(* PLC project Projeto_Silos.project, CODESYS CODESYS V3.5 SP11 Patch 4 *)
(* stored: creationDateTime 2025-10-06T19:54:17.7086948, modificationDateTime 2025-10-06T19:50:28.7209293 *)

PROGRAM PLC_PRG

                    
                  
END_PROGRAM

PROGRAM PRG_Simulacao

                    
                  
END_PROGRAM

PROGRAM PRG_Controle

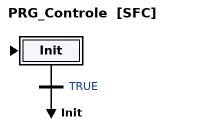
INITIAL_STEP Init:
END_STEP
TRANSITION FROM Init TO Init
  := TRUE;
END_TRANSITION
END_PROGRAM

CONFIGURATION Device
  RESOURCE Application ON PLC
    {attribute 'qualified_only'}
    VAR_GLOBAL  (* GVL_IO *)
      LS_01 : BOOL;  (* Chave fim-de-curso Silo 1. TRUE quando Tripper posicionado. *)
      LS_02 : BOOL;  (* Chave fim-de-curso Silo 2. *)
      LS_03 : BOOL;  (* Chave fim-de-curso Silo 3. *)
      LS_04 : BOOL;  (* Chave fim-de-curso Silo 4. *)
      TR_DIST : REAL;  (* Sensor de distância a laser (metragem) . *)
      WT_01 : REAL;  (* Balança de fluxo interna ao tripper (kg/s) . *)
      TR_FW : BOOL;  (* Acionamento frente do Tripper. *)
      TR_BW : BOOL;  (* Acionamento ré do Tripper. *)
      TR_VEL : REAL;  (* Velocidade de deslocamento do Tripper (m/s) . *)
      M_CT_01 : BOOL;  (* Liga/desliga a correia alimentadora CT-01. *)
      BUZINA : BOOL;  (* Ativa a Buzina para sinalização. *)
    END_VAR
    {attribute 'qualified_only'}
    VAR_GLOBAL  (* GVL_SCADA *)
      LIGA_AUTO : BOOL;  (* Comando de LIGA / DESLIGA executado via SCADA. *)
      EMG : BOOL;  (* Sinalização manual de Emergência via SCADA. *)
      REARME : BOOL;  (* Sinalização manual de Rearme via SCADA. *)
      FV_01 : BOOL;  (* Válvula on-off de descarga Silo 1. *)
      FV_02 : BOOL;  (* Válvula on-off de descarga Silo 2. *)
      FV_03 : BOOL;  (* Válvula on-off de descarga Silo 3. *)
      FV_04 : BOOL;  (* Válvula on-off de descarga Silo 4. *)
      LT_01 : REAL;  (* Sensor de nível Silo 1 (Simulado manualmente via IHM, conforme orientação [cite: 123]). *)
      LT_02 : REAL;  (* Sensor de nível Silo 2 (Simulado manualmente via IHM). *)
      LT_03 : REAL;  (* Sensor de nível Silo 3 (Simulado manualmente via IHM). *)
      LT_04 : REAL;  (* Sensor de nível Silo 4 (Simulado manualmente via IHM). *)
      PESO_SL_01 : REAL;  (* Peso total em toneladas do Silo 1[cite: 94]. *)
      PESO_SL_02 : REAL;  (* Peso total em toneladas do Silo 2. *)
      PESO_SL_03 : REAL;  (* Peso total em toneladas do Silo 3. *)
      PESO_SL_04 : REAL;  (* Peso total em toneladas do Silo 4. *)
      STATUS_FALHA : BOOL;  (* Indica que o CLP entrou em modo FALHA[cite: 64]. *)
      STATUS_EMG : BOOL;  (* Status da Emergência (para Alarme). *)
      POS_TRIPPER : REAL;  (* Posição atual do Tripper para Animação Visual. *)
      FALHA_LS_01 : BOOL;  (* Variáveis para simulação de falha das chaves Fim-de-Curso via IHM [cite: 133] *)
      FALHA_LS_02 : BOOL;
      FALHA_LS_03 : BOOL;
      FALHA_LS_04 : BOOL;
    END_VAR
    TASK Task_Simulacao(INTERVAL := T#20ms, PRIORITY := 10);
    TASK Task_Controle(INTERVAL := T#100ms, PRIORITY := 5);
    PROGRAM PRG_Simulacao WITH Task_Simulacao : PRG_Simulacao;
    PROGRAM PRG_Controle WITH Task_Controle : PRG_Controle;
  END_RESOURCE
END_CONFIGURATION
